FUNCTION_BLOCK FB_TOR_ES EXTENDS FB_TOR_Base
//////////////////
//  Emergency stop system
//////////////////
VAR_INPUT PERSISTENT
	// Parameters of the Object (instance/model specific) 
	ParamTempoEs :TIME:=T#2S;								(* (s) Tempo before raising an alarm*)
END_VAR

VAR_OUTPUT
	//Child objects
	
END_VAR

VAR_INPUT
	// I/O Inputs 		                                     				
		
	
END_VAR

VAR
	//M_ALARMMANAGEMENT VARIABLES//
		FB_PermAlarm				: SR ;					// (NA) FB to maintain emergency stop Alarm 
		TON_ES						: TON ; 
 
	//M_STATEMANAGER VARIABLES//
		MesDataExd			: TOR_Standard ;  	
END_VAR

METHOD M_AlarmManagement
//////////////////
// Manages Smoke detector alarms and warnings
/////////////////

VAR 
	// Method local variables (reinitialized at each cycle) 
	FB_AlarmCodeManager			: FB_AlarmCodeManager ; 
	bAlarmsNbSensors			: BOOL;
END_VAR
// Detection Variables
TON_ES(IN:= MesDataExd.MesData.MesAlarmState , PT:= ParamTempoEs ); 
FB_PermAlarm(SET1 := TON_ES.Q, Reset := CmdClearFault_G OR IN_CmdReset_L); 							// SR FB for keep fire if burn

bAlarmsNbSensors	:= SEL(ParamNbSensors=9,FALSE, IN_MesState1_IO <> IN_MesState2_IO);
// ALARM CODE //
	FB_AlarmCodeManager(
		bAlarm1			:= FB_PermAlarm.Q1,  														// Emergency stop		
		bAlarm2			:= bAlarmsNbSensors, 														// Incoherent measures between sensors
		bAlarm3			:=FALSE, 																	// 
		bAlarm4			:=FALSE, 																	// 
		bAlarm5			:=FALSE, 																	//
		bAlarm6			:=FALSE,                                                                    //
		bAlarm7			:=FALSE,                                                                    //
		bAlarm8			:=FALSE,                                                                    //
		bAlarm9			:=FALSE,                                                                    //
		bAlarm10		:=FALSE,                                                                    //
		bAlarm11		:=FALSE,                                                                    //
		bAlarm12		:=FALSE,                                                                    //
		bAlarm13		:=FALSE,                                                                    //
		bAlarm14		:=FALSE,                                                                    //
		bAlarm15		:=FALSE,                                                                    //
		wAlarmCode		=>MesDataExd.MesData.MesAlarmCode );
		
// WARNING CODE //
	FB_AlarmCodeManager(
		bAlarm1			:=IN_MesState1_IO OR IN_MesState2_IO,	 	 								// At least one detector is ON 
		bAlarm2			:=FALSE, 																	// 
		bAlarm3			:=FALSE, 																	// 
		bAlarm4			:=FALSE, 																	// 
		bAlarm5			:=FALSE, 																	//
		bAlarm6			:=FALSE,                                                                    //
		bAlarm7			:=FALSE,                                                                    //
		bAlarm8			:=FALSE,                                                                    //
		bAlarm9			:=FALSE,                                                                    //
		bAlarm10		:=FALSE,                                                                    //
		bAlarm11		:=FALSE,                                                                    //
		bAlarm12		:=FALSE,                                                                    //
		bAlarm13		:=FALSE,                                                                    //
		bAlarm14		:=FALSE,                                                                    //
		bAlarm15		:=FALSE,                                                                    //
		wAlarmCode		=>MesDataExd.MesData.MesWarningCode);
		
// EVENT CODE //
	FB_AlarmCodeManager(
		bAlarm1			:= IN_MesState1_IO, 														// First sensor is ON
		bAlarm2			:= IN_MesState2_IO, 														// Second sensor is ON
		bAlarm3			:= FALSE, 																	// 
		bAlarm4			:= FALSE, 																	// 
		bAlarm5			:= FALSE, 																	//
		bAlarm6			:= FALSE,                   												//
		bAlarm7			:= FALSE,                   												//
		bAlarm8			:= FALSE,                   												//
		bAlarm9			:= FALSE,                   												//
		bAlarm10		:= FALSE,                   												//
		bAlarm11		:= FALSE,                   												//
		bAlarm12		:= FALSE,                   												//
		bAlarm13		:= FALSE,                   												//
		bAlarm14		:= FALSE,                   												//
		bAlarm15		:= FALSE,                   												//
		wAlarmCode		=>MesDataExd.MesData.MesEventCode);
END_METHOD

METHOD M_Execute
//////////////////
//  Method Calls 
/////////////////

VAR 
	// Method local variables (reinitialized at each cycle) 

END_VAR

	
	IF ParamNbSensors = 9 THEN // Use of contactor bi-stable No and NC
		IN_MesState2_IO := NOT IN_MesState2_IO;
	END_IF
SUPER^.M_Execute() ;
END_METHOD

METHOD M_StateManager
//////////////////
// Detect when fire occurs
/////////////////

VAR 
	// Method local variables (reinitialized at each cycle)
 	MesStateInterm1 : BOOL;
	MesStateInterm2 : BOOL;
END_VAR

IF ParamCableCutSecurity THEN
	MesStateInterm1 := NOT IN_MesState1_IO ; 
	MesStateInterm2 := NOT IN_MesState2_IO ; 
ELSE 
	MesStateInterm1 := IN_MesState1_IO;
	MesStateInterm2 := IN_MesState2_IO;
END_IF

IF ParamNbSensors = 1 THEN 
	MesStateInterm2 :=  MesStateInterm1;
END_IF

IF ParamAtleastOne THEN 
MesDataExd.MesData.MesAlarmState := MesStateInterm1 OR MesStateInterm2 ; 
ELSE
MesDataExd.MesData.MesAlarmState := MesStateInterm1 AND MesStateInterm2 ; 
END_IF

R_TRIGAlarm(CLK:= MesDataExd.MesData.MesAlarmState ) ; 
IF R_TRIGAlarm.Q THEN
	MesCountAlarm :=  MIN(MesCountAlarm + 1 ,4294967295 ) ; 
ELSIF IN_ResetCounter THEN 
	MesCountAlarm := 0 ; 
END_IF

MesDataExd.MesData.MesCountAlarm	:= MesCountAlarm ;
END_METHOD

END_FUNCTION_BLOCK

(* stored: Version 1.1.0.1, ProductVersion 3.1.4024.11
   POU FB_TOR_ES: Id {e91e8373-dcc8-4cd1-acef-c21833e8b897}, SpecialFunc None
   Method M_AlarmManagement: Id {f2b23fb8-4b09-4e33-a613-cbc064696194}
   Method M_Execute: Id {e8e93625-b96d-4c46-997f-834dd56dcf5f}
   Method M_StateManager: Id {97eb67af-5283-4425-b221-a0b4c891515b} *)
